Fanuc KAREL source: kt00066.KL

PROGRAM KT00066
%NOLOCKGROUP
VAR
I1:INTEGER;I2:INTEGER;OUT:REAL
BEGIN
--
--
I1=2
I2=3
I1=2
I2=3
OUT=((I1*I2))
END KT00066
